// TIA Portal V17 export
// export: Created 2026-04-13T11:12:45.126939Z, ExportSetting WithDefaults, DisplayName Totally Integrated Automation Portal, DisplayVersion V17 Update 4, DisplayName TIA Portal Openness, DisplayVersion V17 Update 4, DisplayName TIA Portal Version Control Interface, DisplayVersion V17, DisplayName SINAMICS Startdrive Advanced, DisplayVersion V17, DisplayName SINAMICS Startdrive G130, G150, S120, S150, SINAMICS MV, S210, DisplayVersion V17, DisplayName SINAMICS Startdrive G110M, G120, G120C, G120D, G120P, G115D, DisplayVersion V17, DisplayName STEP 7 Professional, DisplayVersion V17 Update 4, DisplayName STEP 7 Safety, DisplayVersion V17, DisplayName WinCC Professional, DisplayVersion V17 Update 4
VAR_GLOBAL   // PLC tag table "AIQM"
   IWJF进风流量计 AT %MW600 : Int;
   IWJL进料流量 AT %MW602 : Int;
   IWJF进风压差变送器 AT %MW604 : Int;
   IWCF出风高效压差变送器 AT %MW606 : Int;
   IWBD布袋压差变送器 AT %MW608 : Int;
   IWSS输送高效压差变送器 AT %MW610 : Int;
   IWJL进料压力 AT %MW612 : Int;
   IWTN塔内压力 AT %MW614 : Int;
   IWGD管道压力变送器 AT %MW616 : Int;
   IWJD进氮压力 AT %MW618 : Int;
   IWFK放空比例反馈 AT %MW620 : Int;
   IWJF进风加热比例反馈 AT %MW622 : Int;
   IWHF回风加热比例反馈 AT %MW624 : Int;
   IWWH雾化油压 AT %MW626 : Int;
   IWYH氧含仪1 AT %MW628 : Int;
   IWYH氧含仪2 AT %MW630 : Int;
   IWYJ一级溶剂液位计 AT %MW632 : Int;
   IWEJ二级溶剂液位计 AT %MW634 : Int;
   IWCW除雾溶剂液位计 AT %MW636 : Int;
   IWSF送风机 AT %MW638 : Int;
   IWYF引风机 AT %MW640 : Int;
   IWLX离心雾化器 AT %MW642 : Int;
   IWJL进料泵 AT %MW644 : Int;
   QWSF送风机 AT %MW700 : Int;
   QWYF引风机 AT %MW702 : Int;
   QWLX离心雾化器 AT %MW704 : Int;
   QWJL进料泵 AT %MW706 : Int;
   QWFK放空比例调节阀 AT %MW708 : Int;
   QWJF进风加热比例调节阀 AT %MW710 : Int;
   QWHF回风加热比例调节阀 AT %MW712 : Int;
   IWFD阀岛气压 AT %MW646 : Int;
   IWQZ前置水罐液位计 AT %MW648 : Int;
   IWBY备用2 AT %MW650 : Int;
   IWBY备用3 AT %MW652 : Int;
   IWBY备用4 AT %MW654 : Int;
   IWBY备用5 AT %MW656 : Int;
   IWBY备用6 AT %MW658 : Int;
   IWBY备用7 AT %MW660 : Int;
   IWBY备用8 AT %MW662 : Int;
   IWBY备用9 AT %MW664 : Int;
END_VAR
